{attribute 'GeneratedUsingTerminal: EL2535-0000-0016'}
{attribute addProperty BoxType "EL2535-0000-0016"}
{attribute addProperty Id "StatusAT %I*Status_EBCAF3EC5"}
{attribute addProperty CRC "756740928"}
{attribute addProperty Size "5"}
TYPE PWM_Status_Channel_2D1AF340 EXTENDS InputBase_8311D824 :
STRUCT
	{attribute addProperty Name "Status"}
	Status AT %I* : Status_EBCAF3EC;
END_STRUCT
END_TYPE

(* stored: Version 1.2.0.0, ProductVersion 3.1.4024.11
   DUT PWM_Status_Channel_2D1AF340: Id {a5856d66-2034-46b6-8a67-622aa5c8d8c9} *)
